FUNCTION_BLOCK FB_Coordinador_SFC

VAR CONSTANT
LISTA_CONDICIONES: ARRAY[1..TAMANO_LISTA_CONDICIONES] OF CaracteristicasPieza:=[(Claro:=FALSE, Metalico:=FALSE, Alta:=TRUE), //Negra alta
					(Claro:=TRUE,Metalico:=FALSE,Alta:=TRUE), //Blanca alta					
					(Claro:=TRUE, Metalico:=TRUE, Alta:=TRUE), //Metal alta
					(Claro:=FALSE, Metalico:=FALSE, Alta:=FALSE), //Negra baja
					(Claro:=TRUE, Metalico:=FALSE, Alta:=FALSE), //Blanca baja					
					(Claro:=TRUE, Metalico:=TRUE, Alta:=FALSE)]; //Metal baja
END_VAR

VAR_IN_OUT
	ListadePiezas: ARRAY[1..TAMANO_LISTA_PIEZAS] OF Pieza; // Array de tamaño 8 piezas 
	ListaPiezasSolicitadas: ARRAY[1..TAMANO_LISTA_CONDICIONES] OF UINT; // Array de 6 condiciones (blanca, negra y metálica, de momento)
	FaltaMaterial: BOOL;
END_VAR

VAR_INPUT
	  // SFC-Flags
    SFCPause: BOOL;
    SFCReset: BOOL;
    
    // Indicadores de sincronizacion
    Ack: BOOL := TRUE;
    Execute: BOOL;
    
    // Indicadores de control
    Resume: BOOL;
    StepByStep: BOOL;
	FinCiclo: BOOL;
    PiezaAPieza: BOOL;
    // Parametros de sincronizacion
    PaleSituado: BOOL;
	AlimentadorAvanzado: BOOL;
    PiezaCargada: BOOL;
	PlatoEmpujado: BOOL;
	PiezaMedida: BOOL;
    PiezaDescargada: BOOL;
    PiezaRechazada: BOOL;
    PaleTransferido: BOOL;
	PlatoRetrocedido: BOOL;
    
    // Parametros
    CondicionInicial: BOOL;

	//Variables auxiliares
	NCiclos: INT;
	AuxNciclosDesechar: INT := 1;
	AuxNciclosDescargar: INT := 1;
	ListoParaRechazar: BOOL := FALSE;
	ListoParaDescargar: BOOL := FALSE;
	ListoParaMedir: BOOL := FALSE;
	AUX_Suma_Solicitadas: UINT;
	
END_VAR
VAR_OUTPUT
	 // Indicadores de sincronizacion
    Done: BOOL;
    Ready: BOOL;
	Fallo: BOOL;
	FinPieza: BOOL;

    // Parametros de sincronizacion
    SituaPale: BOOL;
	AvanzaAlimentador: BOOL;
	EmpujaPlato: BOOL;
	MedidorMide: BOOL;
    CargaPieza: BOOL;
    DescargaPieza: BOOL;
    RechazaPieza: BOOL;
    TransfierePale: BOOL;
	RetrocederPlato: BOOL;
    
    // Salidas
    LamparaAlarma: BOOL;
    LamparaMarcha: BOOL;
	
	//Variables
	UnidadesSolicitadas: UINT := 1;
	UnidadesPendientes: UINT;
    UnidadesRealizadas: UINT; 
	
END_VAR
VAR

END_VAR

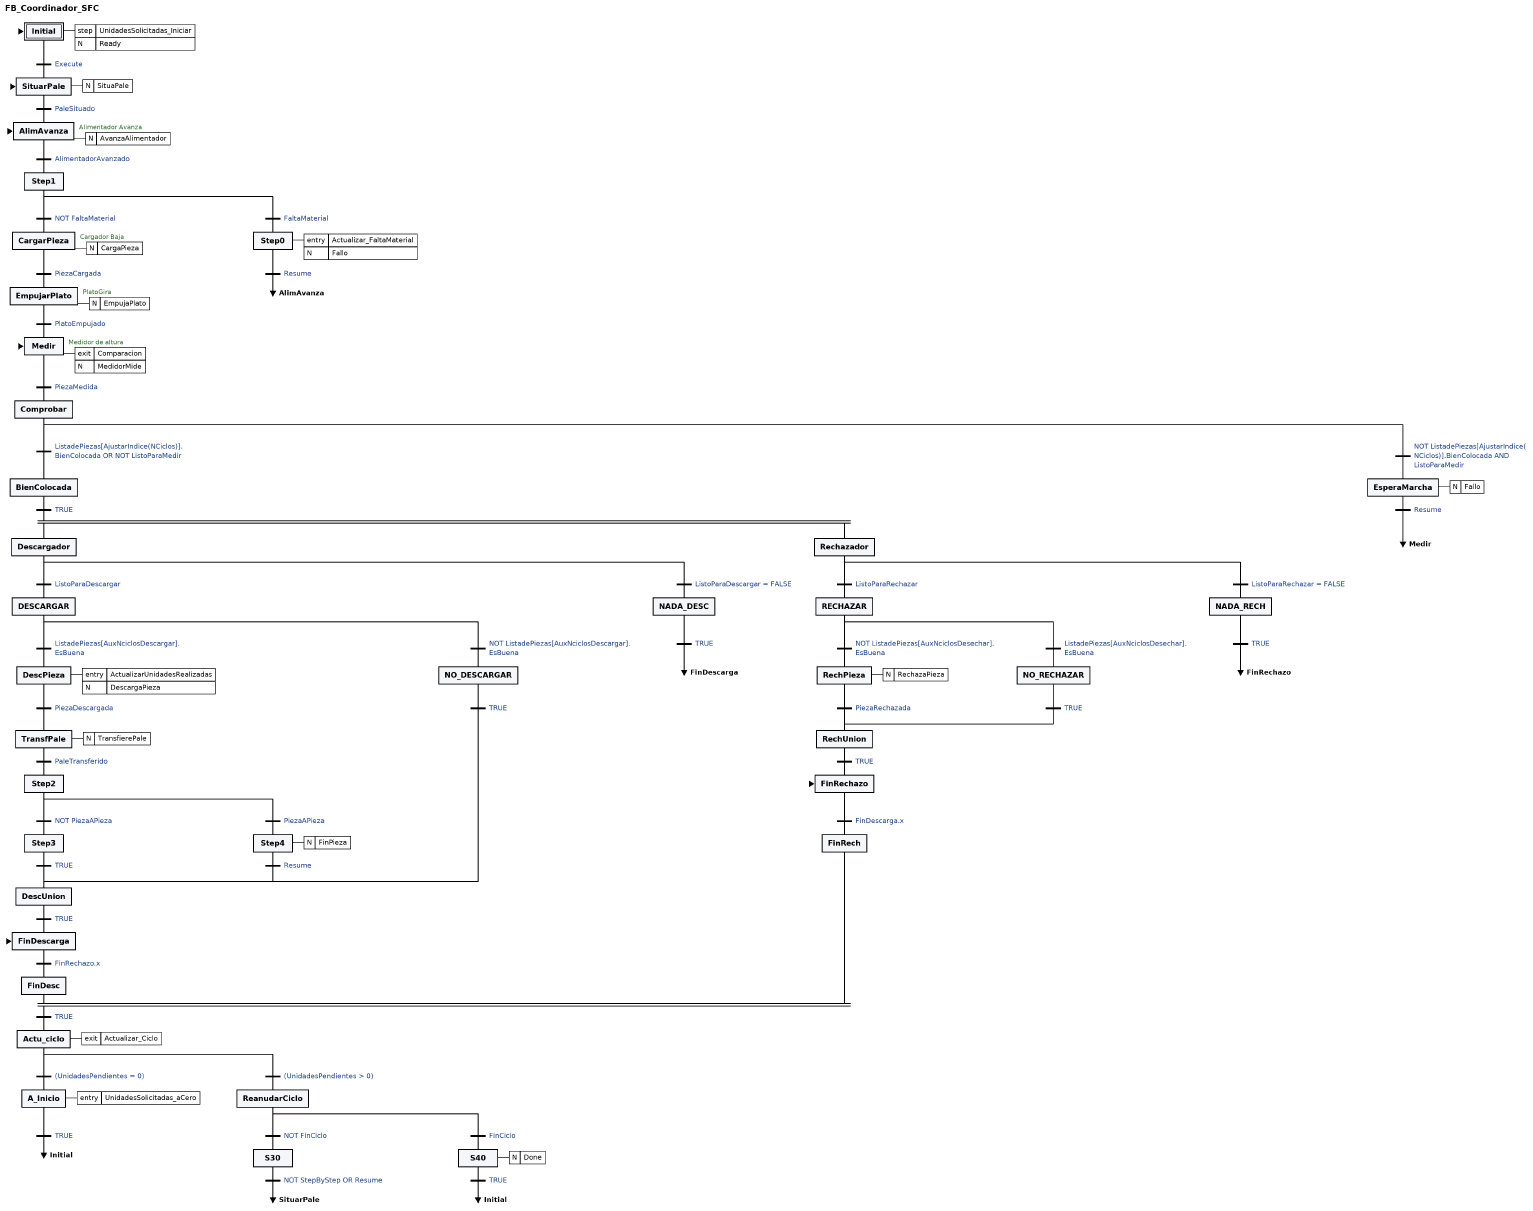
INITIAL_STEP Initial:
    UnidadesSolicitadas_Iniciar(N);  // step action
    Ready(N);
END_STEP
TRANSITION FROM Initial TO SituarPale
    := Execute;
END_TRANSITION
STEP SituarPale:
    SituaPale(N);
END_STEP
TRANSITION FROM SituarPale TO AlimAvanza
    := PaleSituado;
END_TRANSITION
// Alimentador Avanza
STEP AlimAvanza:
    AvanzaAlimentador(N);
END_STEP
TRANSITION FROM AlimAvanza TO Step1
    := AlimentadorAvanzado;
END_TRANSITION
STEP Step1:
END_STEP
TRANSITION FROM Step1 TO CargarPieza
    := NOT FaltaMaterial;
END_TRANSITION
TRANSITION FROM Step1 TO Step0
    := FaltaMaterial;
END_TRANSITION
STEP Step0:
    Actualizar_FaltaMaterial(P1);  // entry action
    Fallo(N);
END_STEP
TRANSITION FROM Step0 TO AlimAvanza
    := Resume;
END_TRANSITION
// Cargador Baja
STEP CargarPieza:
    CargaPieza(N);
END_STEP
TRANSITION FROM CargarPieza TO EmpujarPlato
    := PiezaCargada;
END_TRANSITION
// PlatoGira
STEP EmpujarPlato:
    EmpujaPlato(N);
END_STEP
TRANSITION FROM EmpujarPlato TO Medir
    := PlatoEmpujado;
END_TRANSITION
// Medidor de altura
STEP Medir:
    Comparacion(P0);  // exit action
    MedidorMide(N);
END_STEP
TRANSITION FROM Medir TO Comprobar
    := PiezaMedida;
END_TRANSITION
STEP Comprobar:
END_STEP
TRANSITION FROM Comprobar TO BienColocada
    := ListadePiezas[AjustarIndice(NCiclos)].BienColocada OR NOT ListoParaMedir;
END_TRANSITION
STEP BienColocada:
END_STEP
TRANSITION FROM BienColocada TO (Descargador, Rechazador)
    := TRUE;
END_TRANSITION
TRANSITION FROM Comprobar TO EsperaMarcha
    := NOT ListadePiezas[AjustarIndice(NCiclos)].BienColocada AND ListoParaMedir;
END_TRANSITION
STEP EsperaMarcha:
    Fallo(N);
END_STEP
TRANSITION FROM EsperaMarcha TO Medir
    := Resume;
END_TRANSITION
STEP Descargador:
END_STEP
TRANSITION FROM Descargador TO DESCARGAR
    := ListoParaDescargar;
END_TRANSITION
STEP DESCARGAR:
END_STEP
TRANSITION FROM Descargador TO NADA_DESC
    := ListoParaDescargar = FALSE;
END_TRANSITION
STEP NADA_DESC:
END_STEP
TRANSITION FROM NADA_DESC TO FinDescarga
    := TRUE;
END_TRANSITION
TRANSITION FROM DESCARGAR TO DescPieza
    := ListadePiezas[AuxNciclosDescargar].EsBuena;
END_TRANSITION
STEP DescPieza:
    ActualizarUnidadesRealizadas(P1);  // entry action
    DescargaPieza(N);
END_STEP
TRANSITION FROM DescPieza TO TransfPale
    := PiezaDescargada;
END_TRANSITION
STEP TransfPale:
    TransfierePale(N);
END_STEP
TRANSITION FROM TransfPale TO Step2
    := PaleTransferido;
END_TRANSITION
STEP Step2:
END_STEP
TRANSITION FROM Step2 TO Step3
    := NOT PiezaAPieza;
END_TRANSITION
STEP Step3:
END_STEP
TRANSITION FROM Step3 TO DescUnion
    := TRUE;
END_TRANSITION
TRANSITION FROM Step2 TO Step4
    := PiezaAPieza;
END_TRANSITION
STEP Step4:
    FinPieza(N);
END_STEP
TRANSITION FROM Step4 TO DescUnion
    := Resume;
END_TRANSITION
TRANSITION FROM DESCARGAR TO NO_DESCARGAR
    := NOT ListadePiezas[AuxNciclosDescargar].EsBuena;
END_TRANSITION
STEP NO_DESCARGAR:
END_STEP
TRANSITION FROM NO_DESCARGAR TO DescUnion
    := TRUE;
END_TRANSITION
STEP DescUnion:
END_STEP
TRANSITION FROM DescUnion TO FinDescarga
    := TRUE;
END_TRANSITION
STEP FinDescarga:
END_STEP
TRANSITION FROM FinDescarga TO FinDesc
    := FinRechazo.x;
END_TRANSITION
STEP FinDesc:
END_STEP
STEP Rechazador:
END_STEP
TRANSITION FROM Rechazador TO RECHAZAR
    := ListoParaRechazar;
END_TRANSITION
STEP RECHAZAR:
END_STEP
TRANSITION FROM Rechazador TO NADA_RECH
    := ListoParaRechazar = FALSE;
END_TRANSITION
STEP NADA_RECH:
END_STEP
TRANSITION FROM NADA_RECH TO FinRechazo
    := TRUE;
END_TRANSITION
TRANSITION FROM RECHAZAR TO RechPieza
    := NOT ListadePiezas[AuxNciclosDesechar].EsBuena;
END_TRANSITION
STEP RechPieza:
    RechazaPieza(N);
END_STEP
TRANSITION FROM RechPieza TO RechUnion
    := PiezaRechazada;
END_TRANSITION
TRANSITION FROM RECHAZAR TO NO_RECHAZAR
    := ListadePiezas[AuxNciclosDesechar].EsBuena;
END_TRANSITION
STEP NO_RECHAZAR:
END_STEP
TRANSITION FROM NO_RECHAZAR TO RechUnion
    := TRUE;
END_TRANSITION
STEP RechUnion:
END_STEP
TRANSITION FROM RechUnion TO FinRechazo
    := TRUE;
END_TRANSITION
STEP FinRechazo:
END_STEP
TRANSITION FROM FinRechazo TO FinRech
    := FinDescarga.x;
END_TRANSITION
STEP FinRech:
END_STEP
TRANSITION FROM (FinDesc, FinRech) TO Actu_ciclo
    := TRUE;
END_TRANSITION
STEP Actu_ciclo:
    Actualizar_Ciclo(P0);  // exit action
END_STEP
TRANSITION FROM Actu_ciclo TO A_Inicio
    := (UnidadesPendientes = 0);
END_TRANSITION
TRANSITION FROM Actu_ciclo TO ReanudarCiclo
    := (UnidadesPendientes > 0);
END_TRANSITION
STEP ReanudarCiclo:
END_STEP
TRANSITION FROM ReanudarCiclo TO S30
    := NOT FinCiclo;
END_TRANSITION
STEP S30:
END_STEP
TRANSITION FROM ReanudarCiclo TO S40
    := FinCiclo;
END_TRANSITION
STEP S40:
    Done(N);
END_STEP
TRANSITION FROM S40 TO Initial
    := TRUE;
END_TRANSITION
TRANSITION FROM S30 TO SituarPale
    := NOT StepByStep OR Resume;
END_TRANSITION
STEP A_Inicio:
    UnidadesSolicitadas_aCero(P1);  // entry action
END_STEP
TRANSITION FROM A_Inicio TO Initial
    := TRUE;
END_TRANSITION

ACTION Actualizar_Ciclo:
Nciclos := Nciclos + 1;
IF Nciclos >= 8 THEN // Si da una vuelta entera
   Nciclos := 0;
END_IF


// Tras 6 ciclos, la pieza puede ser desechada
IF Nciclos >= 5 THEN
   ListoParaRechazar := TRUE;
END_IF

// Tras 7 ciclos, la pieza puede ser descargada
IF  Nciclos >= 6 THEN
	ListoParaDescargar := TRUE;
END_IF

ListoParaMedir := TRUE;
END_ACTION

ACTION Actualizar_FaltaMaterial:
FaltaMaterial := FALSE;
END_ACTION

ACTION ActualizarUnidadesRealizadas:
UnidadesRealizadas := UnidadesRealizadas + 1;
UnidadesPendientes := UnidadesPendientes - 1;
END_ACTION

ACTION Comparacion:
//Si esta listo para desechar
IF ListoParaRechazar THEN
   AuxNciclosDesechar := AjustarIndice(Nciclos - 4);
	ListadePiezas[AuxNciclosDesechar].EsBuena := FALSE;
							
	IF ListadePiezas[AuxNciclosDesechar].BienColocada THEN // Evaluacion de las condiciones exigidas
		ListadePiezas[AuxNciclosDesechar].EsBuena := EvaluarPieza(Indice := AuxNciclosDesechar,
																  LISTA_CONDICIONES := LISTA_CONDICIONES,
																  ListadePiezas := ListadePiezas,
																  ListaPiezasSolicitadas := ListaPiezasSolicitadas
																  );
	END_IF
END_IF

//Si esta listo para descargar		
IF ListoParaDescargar THEN	
	AuxNciclosDescargar := AjustarIndice(Nciclos - 5);
END_IF
END_ACTION

METHOD EvaluarPieza : BOOL
VAR_INPUT
	Indice : INT;
	LISTA_CONDICIONES : ARRAY[1..TAMANO_LISTA_CONDICIONES] OF CaracteristicasPieza;
END_VAR

VAR_IN_OUT
	ListadePiezas : ARRAY[1..TAMANO_LISTA_PIEZAS] OF Pieza; 
	ListaPiezasSolicitadas: ARRAY[1..TAMANO_LISTA_CONDICIONES] OF UINT; 
END_VAR

VAR
	ContadorComparacion : INT := 1;
END_VAR
WHILE NOT ListadePiezas[Indice].EsBuena AND ContadorComparacion<7 DO 
	IF ListaPiezasSolicitadas[ContadorComparacion] > 0 THEN 
		IF MEMCMP (ADR(ListadePiezas[Indice].TipoPieza), 
			       ADR(LISTA_CONDICIONES[ContadorComparacion]), 
                   SIZEOF(LISTA_CONDICIONES[ContadorComparacion])) = 0 
       	THEN
			ListadePiezas[Indice].EsBuena := TRUE; 
            ListaPiezasSolicitadas[ContadorComparacion] := ListaPiezasSolicitadas[ContadorComparacion] - 1;
		END_IF
	END_IF
			ContadorComparacion := ContadorComparacion + 1;
END_WHILE

EvaluarPieza := ListadePiezas[Indice].EsBuena;
END_METHOD

ACTION UnidadesSolicitadas_aCero:
ListaPiezasSolicitadas[1] := 0;
ListaPiezasSolicitadas[2] := 0;
ListaPiezasSolicitadas[3] := 0;
ListaPiezasSolicitadas[4] := 0;
ListaPiezasSolicitadas[5] := 0;
ListaPiezasSolicitadas[6] := 0;
END_ACTION

ACTION UnidadesSolicitadas_Iniciar:
UnidadesSolicitadas := 0;
 
//Suma de todas las iezas solicitadas
FOR AUX_Suma_Solicitadas := 1 TO TAMANO_LISTA_CONDICIONES DO
    UnidadesSolicitadas := UnidadesSolicitadas + ListaPiezasSolicitadas[AUX_Suma_Solicitadas];
END_FOR;

    UnidadesPendientes := UnidadesSolicitadas;
END_ACTION

END_FUNCTION_BLOCK

(* stored: Version 1.1.0.1, ProductVersion 3.1.4024.12
   POU FB_Coordinador_SFC: Id {b45996cd-eccc-4c22-9382-c6e15909ae18}, SpecialFunc None
   Folder Acciones: Id {f44a95ce-5ae9-43bf-a768-48c83e9a91a7}
   Folder Metodos: Id {6a678e67-b353-425f-a6a9-6fd80138bb2c}
   Action Actualizar_Ciclo: Id {7672e9a4-1636-48e3-9121-943c79590b09}
   Action Actualizar_FaltaMaterial: Id {952bbbde-0d8d-4917-ac30-cfd32a5de3a5}
   Action ActualizarUnidadesRealizadas: Id {a435d1c6-0c42-453b-9c6b-2f59a6870f2e}
   Action Comparacion: Id {cc2dfffd-ea49-44d6-9229-1803f5153340}
   Method EvaluarPieza: Id {229fa35b-b26f-4178-be0f-17ef1fd8a899}
   Action UnidadesSolicitadas_aCero: Id {a11b1288-f0fc-4a42-8e8e-acc865c04724}
   Action UnidadesSolicitadas_Iniciar: Id {65409e14-37fb-41c0-bf2b-a49448fc8171} *)
